// TIA Portal V14 SP1 export
// export: Created 2019-04-23T05:55:44.1120861Z, ExportSetting WithDefaults, WithReadOnly, DisplayName Totally Integrated Automation Portal, DisplayVersion V14 SP1 Update 6, DisplayName TIA Portal Openness, DisplayVersion V14 SP1 Update 6, DisplayName STEP 7 Professional, DisplayVersion V14 SP1 Update 6, DisplayName WinCC Professional, DisplayVersion V14 SP1 Update 6
FUNCTION_BLOCK "101M2_Compressor_Fan_Motor"   // FB1011, LAD
TITLE = Управление мотором вибратора силоса муки 1 / Управление мотором вентилятора компрессора силоса муки STX1
{ S7_Optimized_Access := 'FALSE' }
VERSION : 0.1
// stored: AutoNumber false, CodeModifiedDate 2019-03-26T07:08:50.1549865Z, CompileDate 2019-03-26T07:08:50.1686584Z, CreationDate 2019-02-04T08:31:08.0295361Z, InterfaceModifiedDate 2019-03-18T05:10:48.624948Z, IsConsistent true, IsIECCheckEnabled false, IsKnowHowProtected false, ISMultiInstanceCapable true, IsWriteProtected false, LibraryConformanceStatus Warning: The object contains access to global data blocks. Warning: The block contains direct access to inputs, outputs, bit memories, indirect access to the registry or indirect access to external memory areas that are unknown at the time of compilation., ModifiedDate 2019-03-26T07:08:50.1549865Z, ParameterModified 2018-04-23T08:12:12.8650856Z, StructureModified 2018-12-26T08:24:27.3403256Z, UDAEnableTagReadback false
   VAR DB_SPECIFIC
      HMI : Struct
         CMD : Struct
            Start : Bool;   // Команда старта вибратора
            Stop : Bool;   // Команда останова вибратора
            Spare_2 : Bool;
            Spare_3 : Bool;
            Spare_4 : Bool;
            Spare_5 : Bool;
            Manual : Bool;   // Ручной режим управления
            Reset_Error : Bool;   // Сброс ошибок
         END_STRUCT;
         DATA : Struct
            StatusWord : Word;   // Слово состояния блока управления мотором
            CntFbkTime : DInt := 1;   // Время контроля включения реле
            TimeDelayOff : DInt := 1200;   // Время задержки отключения мотора вентилятора
         END_STRUCT;
      END_STRUCT;
   END_VAR
   VAR
      One_Motor : "OneMotorManag";
      TON : TON;
   END_VAR
   VAR DB_SPECIFIC
      CntFbkTime : Time;   // Время контроля включения реле
      TimeDelayOff : Time;   // Время задержки отключения мотора вентилятора
      ResetErr : Bool;   // Сброс ошибок / Dumping of errors of the control package
      General_cond_OK : Bool;   // Готовность электрических систем / Conditions of permission of operation of the mechanism are not satisfied
      ManCmd_StartMov : Bool;   // Старт вращения в ручном режиме / Existence of command for rotation of the motor in manual
      ManCmd_StopMov : Bool;   // Стоп вращения в ручном режиме / Existence of command for a stop of rotation of the motor in manual
      AutoCmd_StartMov : Bool;   // Старт вращения в автоматическом режиме / Existence of command for rotation of the motor in the automatic
      AutoCmd_StopMov : Bool;   // Стоп вращения в автоматическом режиме / Existence of command for a stop of rotation of the motor in the automatic
   END_VAR
   VAR_TEMP
      TempBIT : Bool;   // Command 1 on operation of the mechanism in the automatic mode
   END_VAR
   VAR_TEMP   // added for the SCL form of the ladder/FBD networks
      _w1 : Bool;
   END_VAR
BEGIN

REGION Network 1: Сброс ошибок
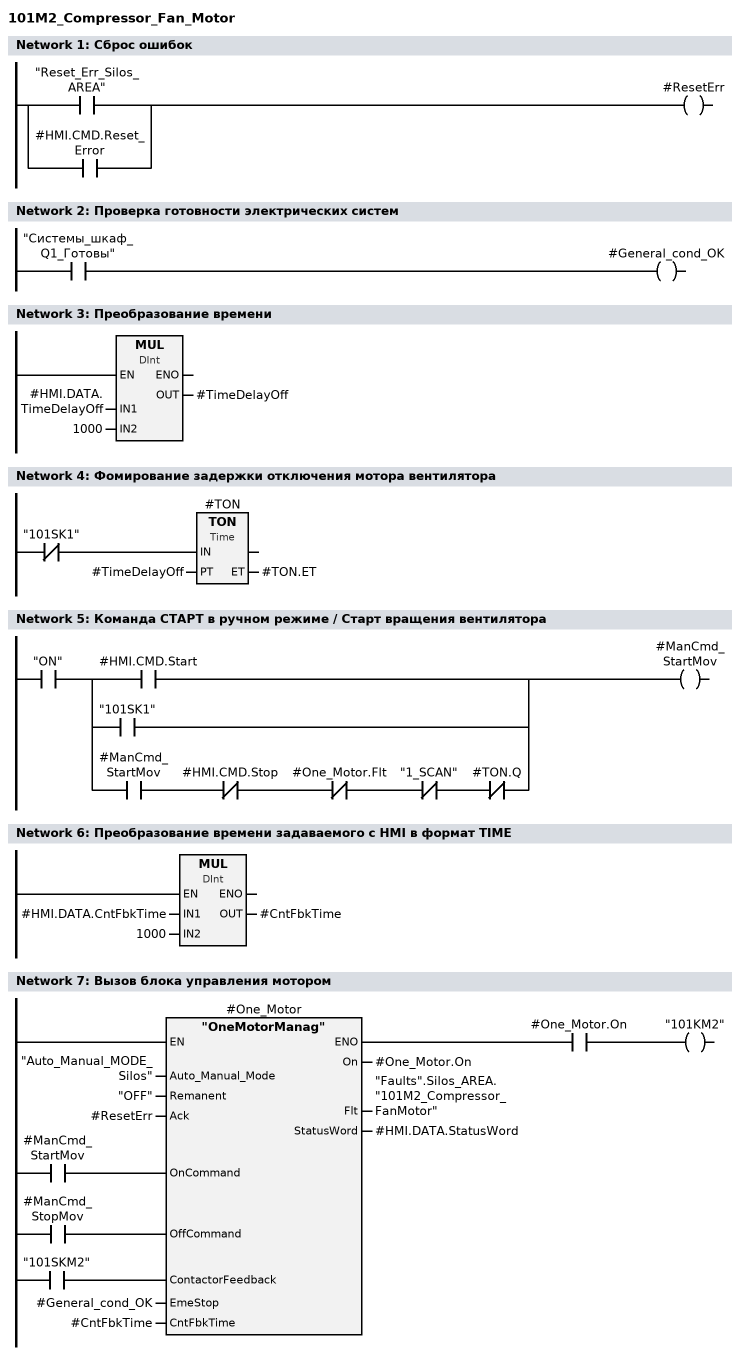
   RUNG wire#powerrail
      Contact( "Reset_Err_Silos_AREA" )
      wire#w1
      Coil( #ResetErr )
   END_RUNG
   RUNG wire#powerrail
      Contact( #HMI.CMD.Reset_Error )
   END_RUNG wire#w1
   // the same network as SCL:
   #ResetErr := "Reset_Err_Silos_AREA" OR #HMI.CMD.Reset_Error;
END_REGION

REGION Network 2: Проверка готовности электрических систем
   RUNG wire#powerrail
      Contact( "Системы_шкаф_Q1_Готовы" )
      Coil( #General_cond_OK )
   END_RUNG
   // the same network as SCL:
   #General_cond_OK := "Системы_шкаф_Q1_Готовы";
END_REGION

REGION Network 3: Преобразование времени
   RUNG wire#powerrail
      { S7_Templates := "SrcType := DInt"; S7_GenerateENO := "TRUE" } Mul(in1 := #HMI.DATA.TimeDelayOff, in2 := 1000, out => #TimeDelayOff)
   END_RUNG
   // the same network as SCL:
   #TimeDelayOff := #HMI.DATA.TimeDelayOff * 1000;
END_REGION

REGION Network 4: Фомирование задержки отключения мотора вентилятора
   RUNG wire#powerrail
      I_Contact( "101SK1" )
      { S7_Templates := "time_type := Time" } #TON.TON(pt := #TimeDelayOff, et => #TON.ET)
   END_RUNG
   // the same network as SCL:
   #TON.TON(IN := NOT "101SK1", PT := #TimeDelayOff, ET => #TON.ET);
END_REGION

REGION Network 5: Команда СТАРТ в ручном режиме / Старт вращения вентилятора
   RUNG wire#powerrail
      Contact( "ON" )
      wire#w1
      Contact( #HMI.CMD.Start )
      wire#w2
      Coil( #ManCmd_StartMov )
   END_RUNG
   RUNG wire#w1
      Contact( "101SK1" )
   END_RUNG wire#w2
   RUNG wire#w1
      Contact( #ManCmd_StartMov )
      I_Contact( #HMI.CMD.Stop )
      I_Contact( #One_Motor.Flt )
      I_Contact( "1_SCAN" )
      I_Contact( #TON.Q )
   END_RUNG wire#w2
   // the same network as SCL:
   #ManCmd_StartMov := "ON" AND (#HMI.CMD.Start OR "101SK1" OR (#ManCmd_StartMov AND NOT #HMI.CMD.Stop AND NOT #One_Motor.Flt AND NOT "1_SCAN" AND NOT #TON.Q));
END_REGION

REGION Network 6: Преобразование времени задаваемого с HMI в формат TIME
   RUNG wire#powerrail
      { S7_Templates := "SrcType := DInt"; S7_GenerateENO := "TRUE" } Mul(in1 := #HMI.DATA.CntFbkTime, in2 := 1000, out => #CntFbkTime)
   END_RUNG
   // the same network as SCL:
   #CntFbkTime := #HMI.DATA.CntFbkTime * 1000;
END_REGION

REGION Network 7: Вызов блока управления мотором
   RUNG wire#powerrail
      #One_Motor(OnCommand := wire#w1, OffCommand := wire#w2, ContactorFeedback := wire#w3, Auto_Manual_Mode := "Auto_Manual_MODE_Silos", Remanent := "OFF", Ack := #ResetErr, EmeStop := #General_cond_OK, CntFbkTime := #CntFbkTime, On => #One_Motor.On, Flt => "Faults".Silos_AREA."101M2_Compressor_FanMotor", StatusWord => #HMI.DATA.StatusWord)
      Contact( #One_Motor.On )
      Coil( "101KM2" )
   END_RUNG
   RUNG wire#powerrail
      Contact( #ManCmd_StartMov )
   END_RUNG wire#w1
   RUNG wire#powerrail
      Contact( #ManCmd_StopMov )
   END_RUNG wire#w2
   RUNG wire#powerrail
      Contact( "101SKM2" )
   END_RUNG wire#w3
   // the same network as SCL:
   #One_Motor(Auto_Manual_Mode := "Auto_Manual_MODE_Silos",   // "OneMotorManag"
              Remanent := "OFF",
              Ack := #ResetErr,
              OnCommand := #ManCmd_StartMov,
              OffCommand := #ManCmd_StopMov,
              ContactorFeedback := "101SKM2",
              EmeStop := #General_cond_OK,
              CntFbkTime := #CntFbkTime,
              On => #One_Motor.On,
              Flt => "Faults".Silos_AREA."101M2_Compressor_FanMotor",
              StatusWord => #HMI.DATA.StatusWord,
              ENO => #_w1);
   "101KM2" := #_w1 AND #One_Motor.On;
END_REGION
END_FUNCTION_BLOCK
